{region '#Template'}
	{attribute 'Version' := '5.1.0.0'}
	{attribute 'Tags' := '"LCID": "1031", "Text": "Gebäudeautomation, Kommunikation, Server, Client, Publisher, Subscriber"'}
	{attribute 'Tags' := '"LCID": "1033", "Text": "Building automation, Communication, Server, Client, Publisher, Subscriber"'}
	{attribute 'Using' := '"Type": "Template", "URI": "Site"'}
	{attribute 'Description' := '"LCID": "1031", "Text": "Server Datenkommunikation"'}
	{attribute 'Description' := '"LCID": "1033", "Text": "Server data communication"'}
{endregion}

FUNCTION_BLOCK FB_BA_AdsComServer_Basic
VAR_INPUT CONSTANT
	WeatherStation			: FB_BA_RawPublisher;
	GeneralSettings			: FB_BA_RawPublisher;
    BuildingAlarms			: FB_BA_RawPublisher;
END_VAR

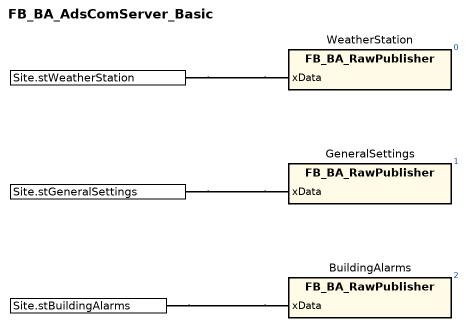
WeatherStation(xData := Site.stWeatherStation); // FB_BA_RawPublisher
GeneralSettings(xData := Site.stGeneralSettings); // FB_BA_RawPublisher
BuildingAlarms(xData := Site.stBuildingAlarms); // FB_BA_RawPublisher

END_FUNCTION_BLOCK

(* stored: Version 1.1.0.1, ProductVersion 3.1.4024.12
   POU FB_BA_AdsComServer_Basic: Id {f35983cf-e8c1-45a3-b7e2-f6836dd5f09f}, SpecialFunc None *)
